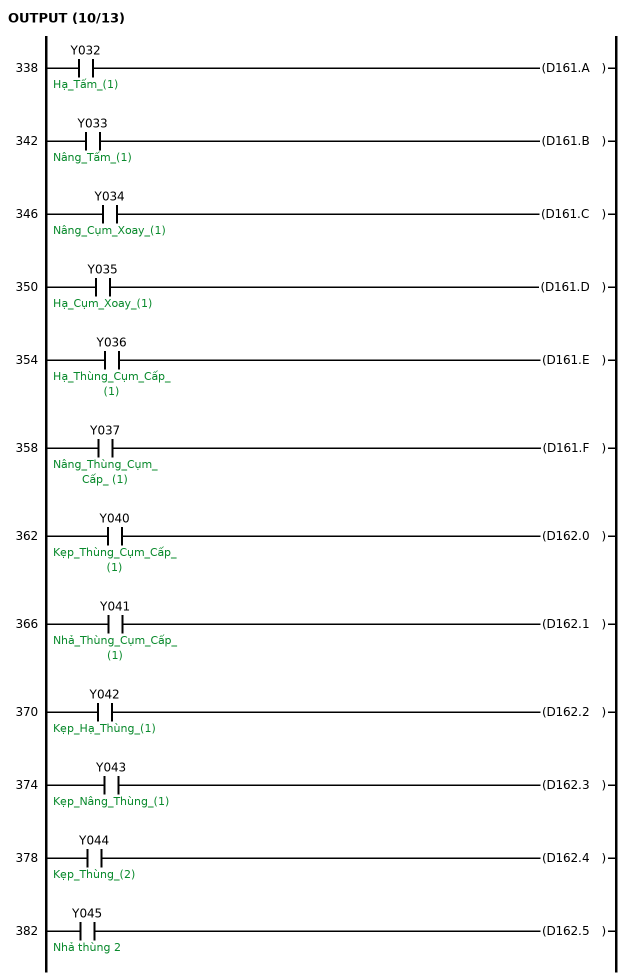
[picture p48: ladder of OUTPUT, rungs at steps 338 to 382]
338   LD      Y032  ; Hạ_Tấm_(1)
      OUT     D161.A
342   LD      Y033  ; Nâng_Tấm_(1)
      OUT     D161.B
346   LD      Y034  ; Nâng_Cụm_Xoay_(1)
      OUT     D161.C
350   LD      Y035  ; Hạ_Cụm_Xoay_(1)
      OUT     D161.D
354   LD      Y036  ; Hạ_Thùng_Cụm_Cấp_ (1)
      OUT     D161.E
358   LD      Y037  ; Nâng_Thùng_Cụm_Cấp_ (1)
      OUT     D161.F
362   LD      Y040  ; Kẹp_Thùng_Cụm_Cấp_(1)
      OUT     D162.0
366   LD      Y041  ; Nhả_Thùng_Cụm_Cấp_(1)
      OUT     D162.1
370   LD      Y042  ; Kẹp_Hạ_Thùng_(1)
      OUT     D162.2
374   LD      Y043  ; Kẹp_Nâng_Thùng_(1)
      OUT     D162.3
378   LD      Y044  ; Kẹp_Thùng_(2)
      OUT     D162.4
382   LD      Y045  ; Nhả thùng 2
      OUT     D162.5
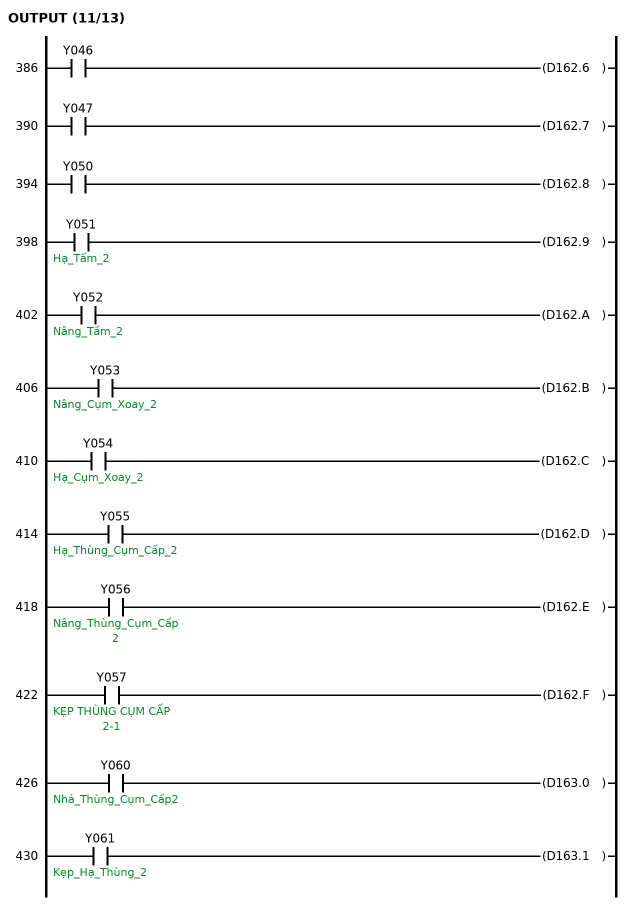
386   LD      Y046
      OUT     D162.6
390   LD      Y047
      OUT     D162.7
394   LD      Y050
      OUT     D162.8
398   LD      Y051  ; Hạ_Tấm_2
      OUT     D162.9
402   LD      Y052  ; Nâng_Tấm_2
      OUT     D162.A
406   LD      Y053  ; Nâng_Cụm_Xoay_2
      OUT     D162.B
410   LD      Y054  ; Hạ_Cụm_Xoay_2
      OUT     D162.C
414   LD      Y055  ; Hạ_Thùng_Cụm_Cấp_2
      OUT     D162.D
418   LD      Y056  ; Nâng_Thùng_Cụm_Cấp 2
      OUT     D162.E
422   LD      Y057  ; KẸP THÙNG CỤM CẤP 2-1
      OUT     D162.F
426   LD      Y060  ; Nhả_Thùng_Cụm_Cấp2
      OUT     D163.0
430   LD      Y061  ; Kẹp_Hạ_Thùng_2
      OUT     D163.1
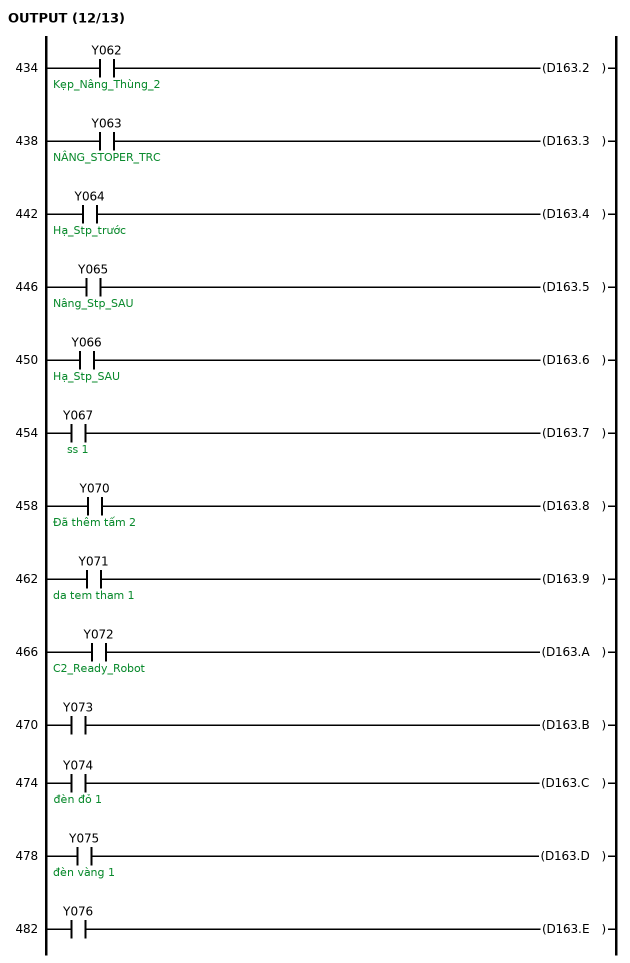
434   LD      Y062  ; Kẹp_Nâng_Thùng_2
      OUT     D163.2
438   LD      Y063  ; NÂNG_STOPER_TRC
      OUT     D163.3
442   LD      Y064  ; Hạ_Stp_trước
      OUT     D163.4
446   LD      Y065  ; Nâng_Stp_SAU
      OUT     D163.5
450   LD      Y066  ; Hạ_Stp_SAU
      OUT     D163.6
454   LD      Y067  ; ss 1
      OUT     D163.7
458   LD      Y070  ; Đã thêm tấm 2
      OUT     D163.8
462   LD      Y071  ; da tem tham 1
      OUT     D163.9
466   LD      Y072  ; C2_Ready_Robot
      OUT     D163.A
470   LD      Y073
      OUT     D163.B
474   LD      Y074  ; đèn đỏ 1
      OUT     D163.C
478   LD      Y075  ; đèn vàng 1
      OUT     D163.D
482   LD      Y076
      OUT     D163.E
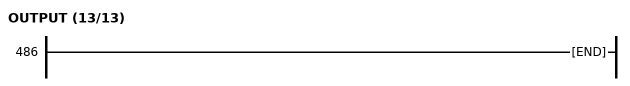
486   END
END_PROGRAM

PROGRAM PC_Ctrl
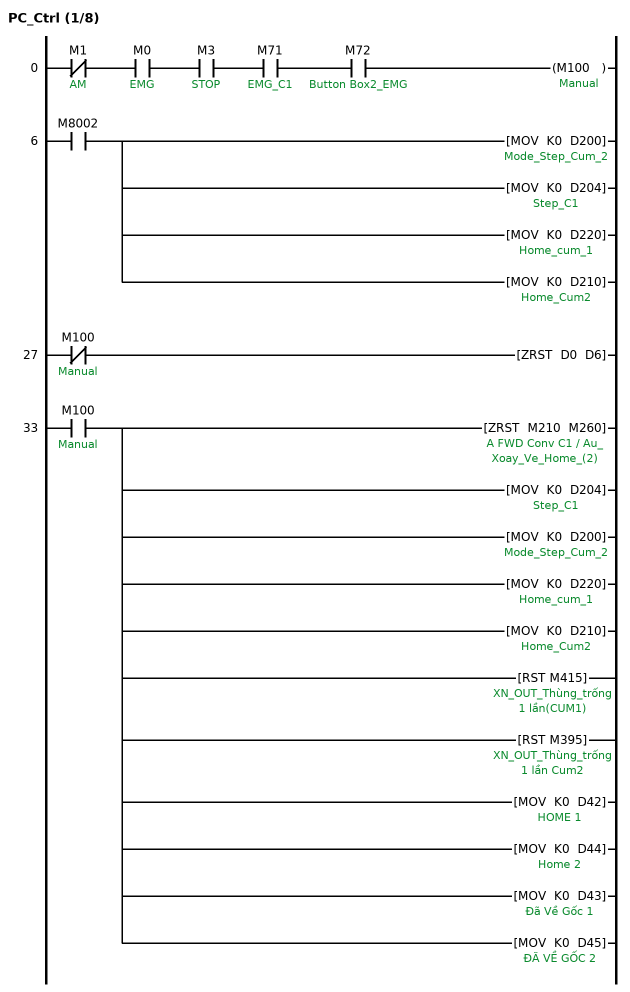
0     LDI     M1  ; AM
      AND     M0  ; EMG
      AND     M3  ; STOP
      AND     M71  ; EMG_C1
      AND     M72  ; Button Box2_EMG
      OUT     M100  ; Manual
6     LD      M8002
      MOV     K0 D200  ; Mode_Step_Cum_2
      MOV     K0 D204  ; Step_C1
      MOV     K0 D220  ; Home_cum_1
      MOV     K0 D210  ; Home_Cum2
27    LDI     M100  ; Manual
      ZRST    D0 D6
33    LD      M100  ; Manual
      ZRST    M210 M260  ; A FWD Conv C1 / Au_ Xoay_Ve_Home_(2)
      MOV     K0 D204
      MOV     K0 D200
      MOV     K0 D220
      MOV     K0 D210
      RST     M415  ; XN_OUT_Thùng_trống 1 lần(CUM1)
      RST     M395  ; XN_OUT_Thùng_trống 1 lần Cum2
      MOV     K0 D42  ; HOME 1
      MOV     K0 D44  ; Home 2
      MOV     K0 D43  ; Đã Về Gốc 1
      MOV     K0 D45  ; ĐÃ VỀ GỐC 2
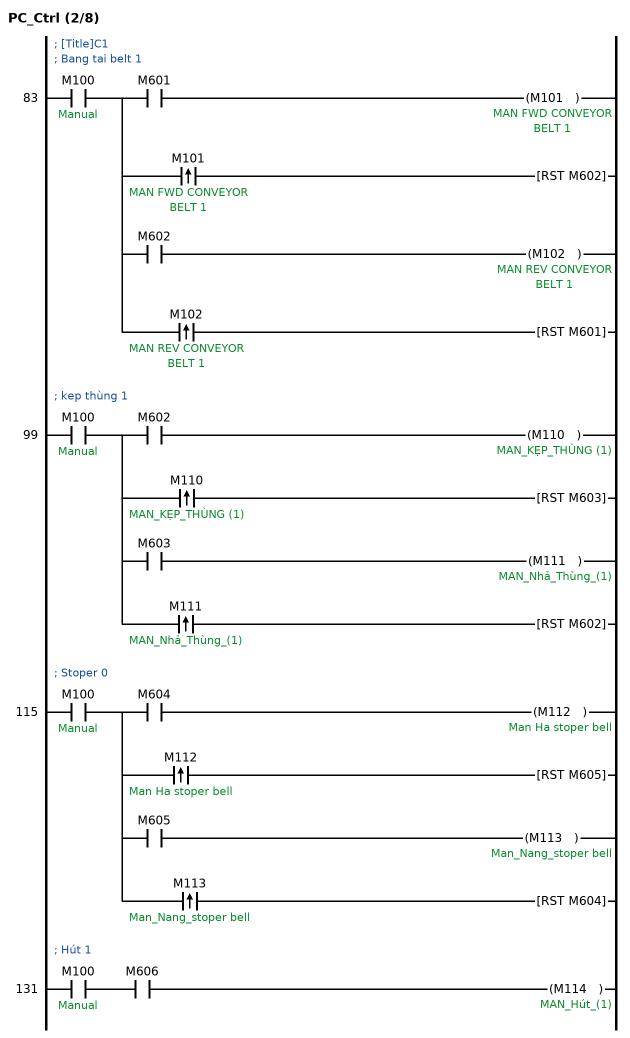
; [Title]C1
; Bang tai belt 1
83    LD      M100  ; Manual
      MPS
      AND     M601
      OUT     M101  ; MAN FWD CONVEYOR BELT 1
      MRD
      ANDP    M101  ; MAN FWD CONVEYOR BELT 1
      RST     M602
      MRD
      AND     M602
      OUT     M102  ; MAN REV CONVEYOR BELT 1
      MPP
      ANDP    M102  ; MAN REV CONVEYOR BELT 1
      RST     M601
; kep thùng 1
99    LD      M100  ; Manual
      MPS
      AND     M602
      OUT     M110  ; MAN_KẸP_THÙNG (1)
      MRD
      ANDP    M110  ; MAN_KẸP_THÙNG (1)
      RST     M603
      MRD
      AND     M603
      OUT     M111  ; MAN_Nhả_Thùng_(1)
      MPP
      ANDP    M111  ; MAN_Nhả_Thùng_(1)
      RST     M602
; Stoper 0
115   LD      M100  ; Manual
      MPS
      AND     M604
      OUT     M112  ; Man Ha stoper bell
      MRD
      ANDP    M112  ; Man Ha stoper bell
      RST     M605
      MRD
      AND     M605
      OUT     M113  ; Man_Nang_stoper bell
      MPP
      ANDP    M113  ; Man_Nang_stoper bell
      RST     M604
; Hút 1
131   LD      M100  ; Manual
      AND     M606
      OUT     M114  ; MAN_Hút_(1)
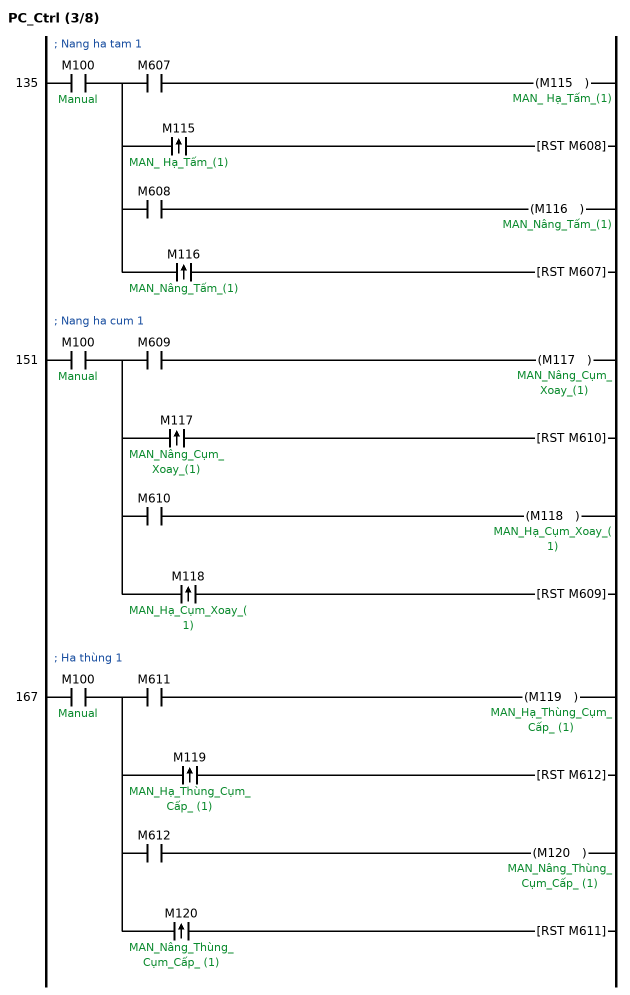
; Nang ha tam 1
135   LD      M100  ; Manual
      MPS
      AND     M607
      OUT     M115  ; MAN_ Hạ_Tấm_(1)
      MRD
      ANDP    M115  ; MAN_ Hạ_Tấm_(1)
      RST     M608
      MRD
      AND     M608
      OUT     M116  ; MAN_Nâng_Tấm_(1)
      MPP
      ANDP    M116  ; MAN_Nâng_Tấm_(1)
      RST     M607
; Nang ha cum 1
151   LD      M100  ; Manual
      MPS
      AND     M609
      OUT     M117  ; MAN_Nâng_Cụm_Xoay_(1)
      MRD
      ANDP    M117  ; MAN_Nâng_Cụm_Xoay_(1)
      RST     M610
      MRD
      AND     M610
      OUT     M118  ; MAN_Hạ_Cụm_Xoay_(1)
      MPP
      ANDP    M118  ; MAN_Hạ_Cụm_Xoay_(1)
      RST     M609
; Ha thùng 1
167   LD      M100  ; Manual
      MPS
      AND     M611
      OUT     M119  ; MAN_Hạ_Thùng_Cụm_Cấp_ (1)
      MRD
      ANDP    M119  ; MAN_Hạ_Thùng_Cụm_Cấp_ (1)
      RST     M612
      MRD
      AND     M612
      OUT     M120  ; MAN_Nâng_Thùng_Cụm_Cấp_ (1)
      MPP
      ANDP    M120  ; MAN_Nâng_Thùng_Cụm_Cấp_ (1)
      RST     M611
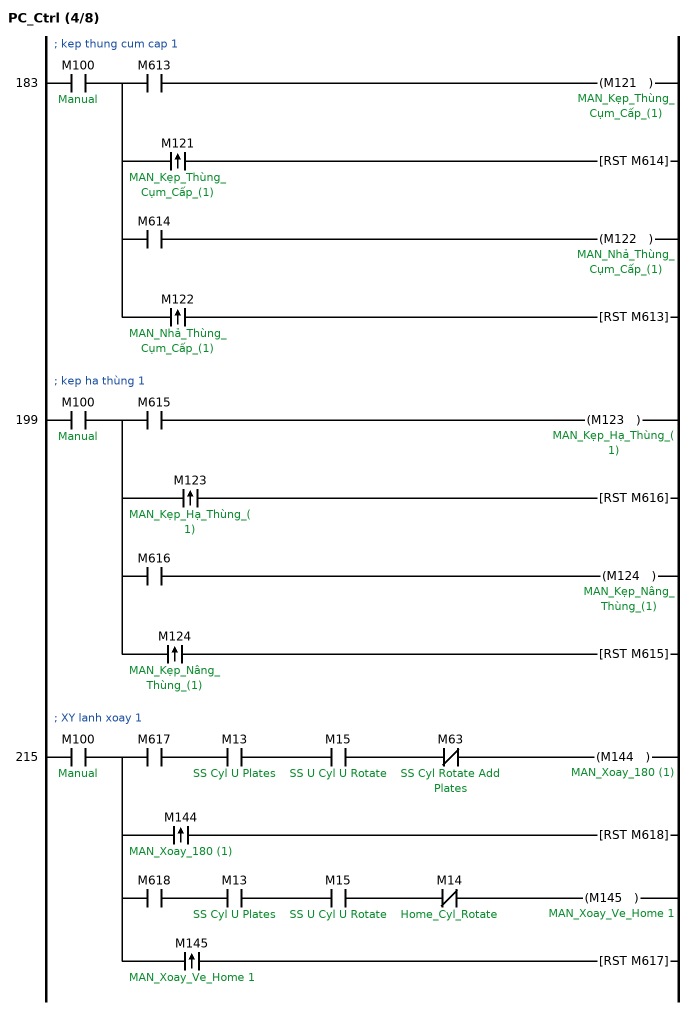
; kep thung cum cap 1
183   LD      M100  ; Manual
      MPS
      AND     M613
      OUT     M121  ; MAN_Kẹp_Thùng_Cụm_Cấp_(1)
      MRD
      ANDP    M121  ; MAN_Kẹp_Thùng_Cụm_Cấp_(1)
      RST     M614
      MRD
      AND     M614
      OUT     M122  ; MAN_Nhả_Thùng_Cụm_Cấp_(1)
      MPP
      ANDP    M122  ; MAN_Nhả_Thùng_Cụm_Cấp_(1)
      RST     M613
; kep ha thùng 1
199   LD      M100  ; Manual
      MPS
      AND     M615
      OUT     M123  ; MAN_Kẹp_Hạ_Thùng_(1)
      MRD
      ANDP    M123  ; MAN_Kẹp_Hạ_Thùng_(1)
      RST     M616
      MRD
      AND     M616
      OUT     M124  ; MAN_Kẹp_Nâng_Thùng_(1)
      MPP
      ANDP    M124  ; MAN_Kẹp_Nâng_Thùng_(1)
      RST     M615
; XY lanh xoay 1
215   LD      M100  ; Manual
      MPS
      AND     M617
      AND     M13  ; SS Cyl U Plates
      AND     M15  ; SS U Cyl U Rotate
      ANI     M63  ; SS Cyl Rotate Add Plates
      OUT     M144  ; MAN_Xoay_180 (1)
      MRD
      ANDP    M144  ; MAN_Xoay_180 (1)
      RST     M618
      MRD
      AND     M618
      AND     M13  ; SS Cyl U Plates
      AND     M15  ; SS U Cyl U Rotate
      ANI     M14  ; Home_Cyl_Rotate
      OUT     M145  ; MAN_Xoay_Ve_Home 1
      MPP
      ANDP    M145  ; MAN_Xoay_Ve_Home 1
      RST     M617
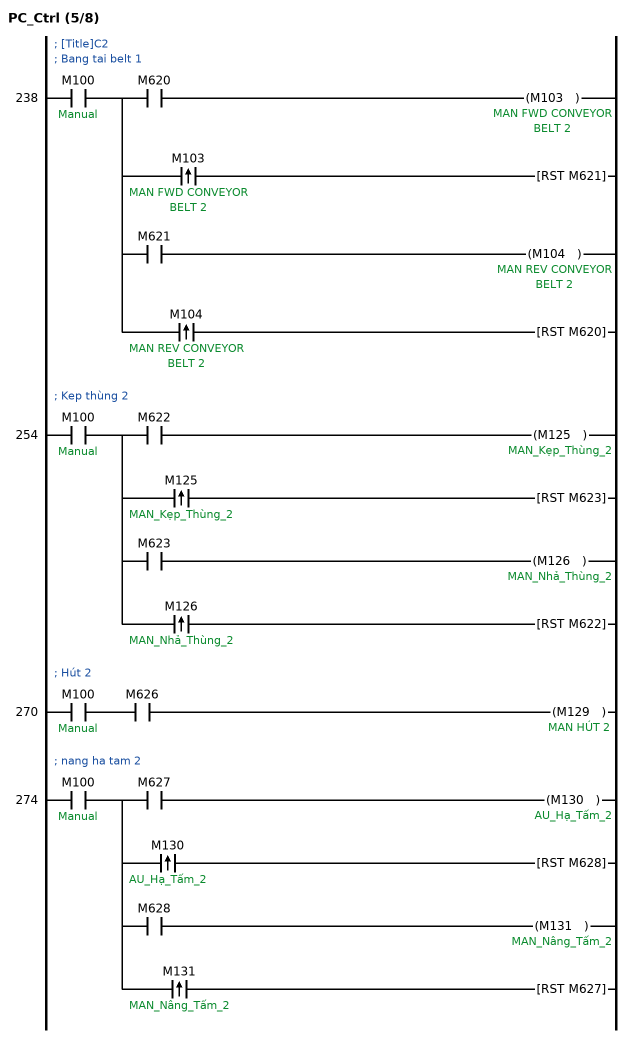
; [Title]C2
; Bang tai belt 1
238   LD      M100  ; Manual
      MPS
      AND     M620
      OUT     M103  ; MAN FWD CONVEYOR BELT 2
      MRD
      ANDP    M103  ; MAN FWD CONVEYOR BELT 2
      RST     M621
      MRD
      AND     M621
      OUT     M104  ; MAN REV CONVEYOR BELT 2
      MPP
      ANDP    M104  ; MAN REV CONVEYOR BELT 2
      RST     M620
; Kep thùng 2
254   LD      M100  ; Manual
      MPS
      AND     M622
      OUT     M125  ; MAN_Kẹp_Thùng_2
      MRD
      ANDP    M125  ; MAN_Kẹp_Thùng_2
      RST     M623
      MRD
      AND     M623
      OUT     M126  ; MAN_Nhả_Thùng_2
      MPP
      ANDP    M126  ; MAN_Nhả_Thùng_2
      RST     M622
; Hút 2
270   LD      M100  ; Manual
      AND     M626
      OUT     M129  ; MAN HÚT 2
; nang ha tam 2
274   LD      M100  ; Manual
      MPS
      AND     M627
      OUT     M130  ; AU_Hạ_Tấm_2
      MRD
      ANDP    M130  ; AU_Hạ_Tấm_2
      RST     M628
      MRD
      AND     M628
      OUT     M131  ; MAN_Nâng_Tấm_2
      MPP
      ANDP    M131  ; MAN_Nâng_Tấm_2
      RST     M627
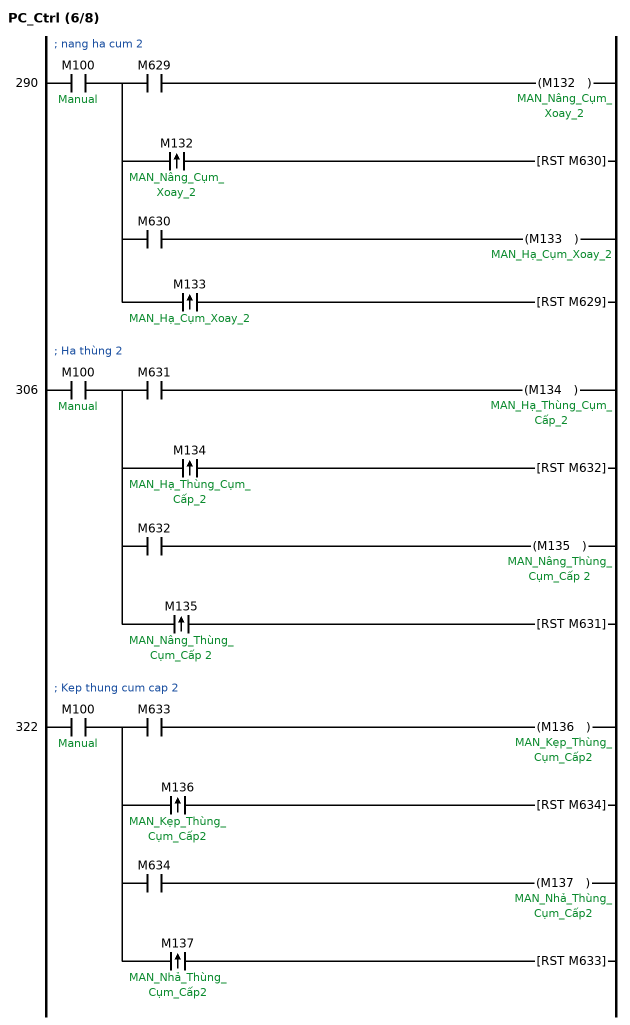
; nang ha cum 2
290   LD      M100  ; Manual
      MPS
      AND     M629
      OUT     M132  ; MAN_Nâng_Cụm_Xoay_2
      MRD
      ANDP    M132  ; MAN_Nâng_Cụm_Xoay_2
      RST     M630
      MRD
      AND     M630
      OUT     M133  ; MAN_Hạ_Cụm_Xoay_2
      MPP
      ANDP    M133  ; MAN_Hạ_Cụm_Xoay_2
      RST     M629
; Ha thùng 2
306   LD      M100  ; Manual
      MPS
      AND     M631
      OUT     M134  ; MAN_Hạ_Thùng_Cụm_Cấp_2
      MRD
      ANDP    M134  ; MAN_Hạ_Thùng_Cụm_Cấp_2
      RST     M632
      MRD
      AND     M632
      OUT     M135  ; MAN_Nâng_Thùng_Cụm_Cấp 2
      MPP
      ANDP    M135  ; MAN_Nâng_Thùng_Cụm_Cấp 2
      RST     M631
; Kep thung cum cap 2
322   LD      M100  ; Manual
      MPS
      AND     M633
      OUT     M136  ; MAN_Kẹp_Thùng_Cụm_Cấp2
      MRD
      ANDP    M136  ; MAN_Kẹp_Thùng_Cụm_Cấp2
      RST     M634
      MRD
      AND     M634
      OUT     M137  ; MAN_Nhả_Thùng_Cụm_Cấp2
      MPP
      ANDP    M137  ; MAN_Nhả_Thùng_Cụm_Cấp2
      RST     M633
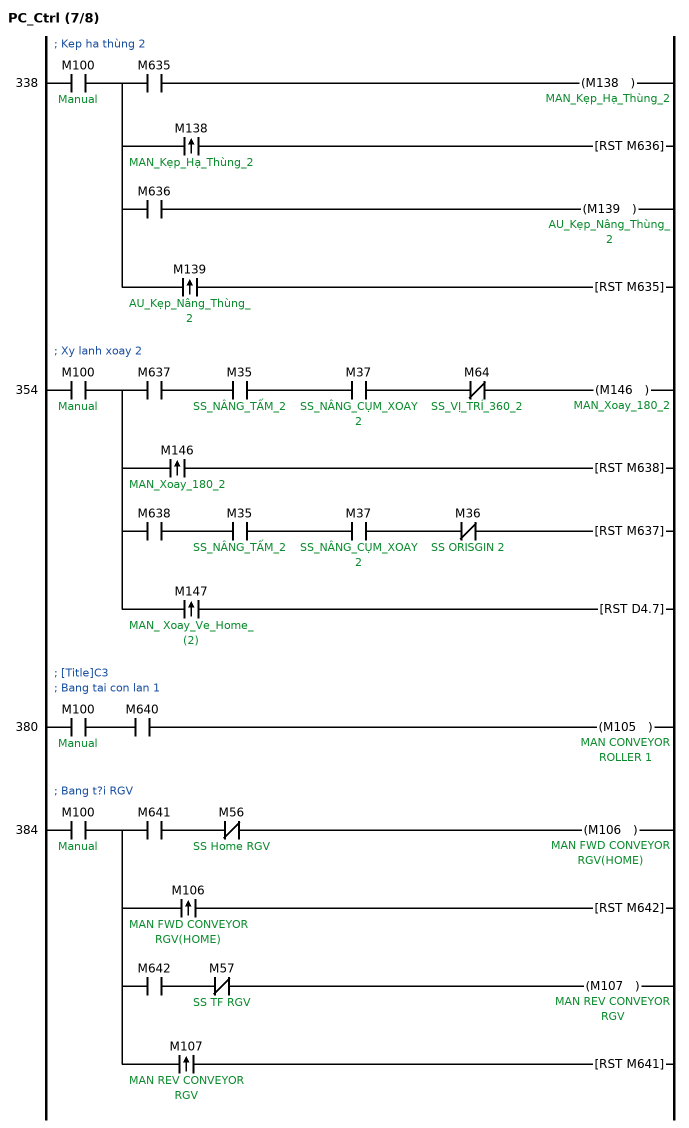
; Kep ha thùng 2
338   LD      M100  ; Manual
      MPS
      AND     M635
      OUT     M138  ; MAN_Kẹp_Hạ_Thùng_2
      MRD
      ANDP    M138  ; MAN_Kẹp_Hạ_Thùng_2
      RST     M636
      MRD
      AND     M636
      OUT     M139  ; AU_Kẹp_Nâng_Thùng_2
      MPP
      ANDP    M139  ; AU_Kẹp_Nâng_Thùng_2
      RST     M635
; Xy lanh xoay 2
354   LD      M100  ; Manual
      MPS
      AND     M637
      AND     M35  ; SS_NÂNG_TẤM_2
      AND     M37  ; SS_NÂNG_CỤM_XOAY 2
      ANI     M64  ; SS_VỊ_TRÍ_360_2
      OUT     M146  ; MAN_Xoay_180_2
      MRD
      ANDP    M146  ; MAN_Xoay_180_2
      RST     M638
      MRD
      AND     M638
      AND     M35  ; SS_NÂNG_TẤM_2
      AND     M37  ; SS_NÂNG_CỤM_XOAY 2
      ANI     M36  ; SS ORISGIN 2
      RST     M637
      MPP
      ANDP    M147  ; MAN_ Xoay_Ve_Home_(2)
      RST     D4.7
; [Title]C3
; Bang tai con lan 1
; 
380   LD      M100  ; Manual
      AND     M640
      OUT     M105  ; MAN CONVEYOR ROLLER 1
; Bang t?i RGV
384   LD      M100  ; Manual
      MPS
      AND     M641
      ANI     M56  ; SS Home RGV
      OUT     M106  ; MAN FWD CONVEYOR RGV(HOME)
      MRD
      ANDP    M106  ; MAN FWD CONVEYOR RGV(HOME)
      RST     M642
      MRD
      AND     M642
      ANI     M57  ; SS TF RGV
      OUT     M107  ; MAN REV CONVEYOR RGV
      MPP
      ANDP    M107  ; MAN REV CONVEYOR RGV
      RST     M641
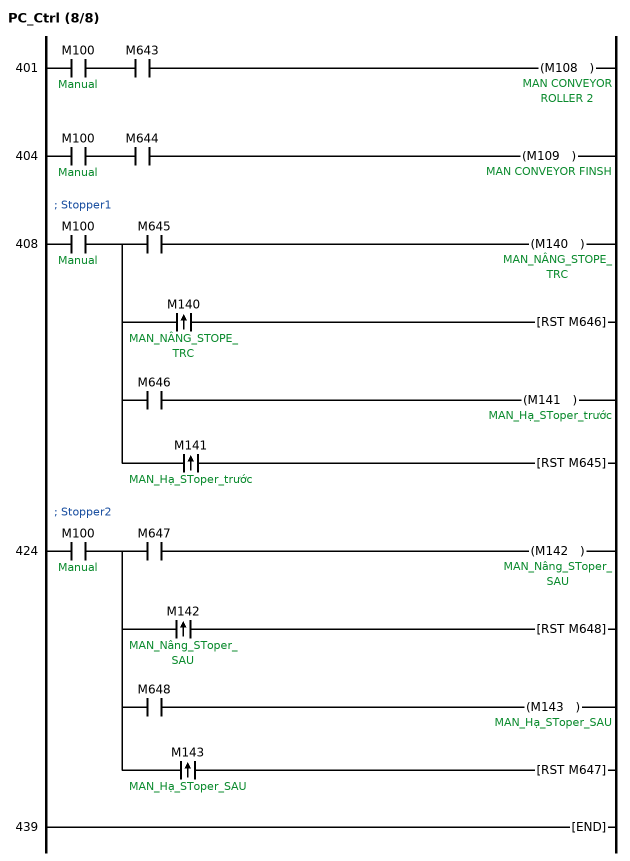
401   LD      M100  ; Manual
      AND     M643
      OUT     M108  ; MAN CONVEYOR ROLLER 2
404   LD      M100  ; Manual
      AND     M644
      OUT     M109  ; MAN CONVEYOR FINSH
; Stopper1
408   LD      M100  ; Manual
      MPS
      AND     M645
      OUT     M140  ; MAN_NÂNG_STOPE_TRC
      MRD
      ANDP    M140  ; MAN_NÂNG_STOPE_TRC
      RST     M646
      MRD
      AND     M646
      OUT     M141  ; MAN_Hạ_SToper_trước
      MPP
      ANDP    M141  ; MAN_Hạ_SToper_trước
      RST     M645
; Stopper2
424   LD      M100  ; Manual
      MPS
      AND     M647
      OUT     M142  ; MAN_Nâng_SToper_SAU
      MRD
      ANDP    M142  ; MAN_Nâng_SToper_SAU
      RST     M648
      MRD
      AND     M648
      OUT     M143  ; MAN_Hạ_SToper_SAU
      MPP
      ANDP    M143  ; MAN_Hạ_SToper_SAU
      RST     M647
439   END
END_PROGRAM

// device comments not shown above
M150  ; MAN 1
M151  ; MAN2
M180  ; HOME
M181  ; HOME 1
M182  ; HOME 2
M195  ; TG STOP
M196  ; NGAT HUT 1
M197  ; NGAT HUT 2
M198  ; TG TRA HANG 2
M199  ; TG TRA HANG 1
M200  ; AUTO
M203  ; Tạm dừng 1
M205  ; HMI_AUTO1
M206  ; HMI_AUTO2
M301  ; TG CHECK VỊ TRÍ LẤY TẤM 1
M302  ; TG CHECK GỐC 1
M303  ; Thêm tấm 1
M305  ; OFF HÚT 1
M306  ; TG TIMER DELAY STOPPER
M310  ; ATUO_SERVO 2 QUAY 180
M311  ; TG CHECK VỊ TRÍ LẤY TẤM 2
M312  ; TG CHECK GỐC 2
M313  ; Thêm tấm 2
M315  ; OFF HÚT 2
M322  ; SS hàng 1 tam (2) va da thêm tam
M326  ; Sansang hang 1 cum
M335  ; KHÓA TAY XOAY 2
M350  ; Req_Add_Plate_C1
M385  ; Home_cum2
M386  ; Bit_Home1
M397  ; Bit_XN_da_xoay_Manual(Cum2)
M399  ; Hang 2 tam
M410  ; Bit_XN_da_xoay_Manual(Cum2)
D1  ; Man_Device_Cum1
D2  ; MAN Device cum1
D3  ; Man Device cum2
D4  ; Man Device cum2
D5  ; MAN Device Cum2
D7  ; MAN HẠ THÙNG 1
D8  ; MAN KẸP THÙNG CỤM CẤP 1
D9  ; MAN KẸP HẠ THÙNG 1
D10  ; XY LANK XOAY1
D11  ; MAN CONVEYOR BELT 2
D12  ; MAN KẸP THÙNG 2
D13  ; MAN KẸP TẤM 2
D14  ; MAN HÚT 2
D15  ; MAN NÂNG HẠ TẤM 2-1
D16  ; MAN NÂNG HẠ CỤM 2
D17  ; MAN HẠ THÙNG 2
D18  ; MAN KẸP THÙNG CỤM CẤP 2
D19  ; MAN KẸP HẠ THÙNG 2
D20  ; XY LANK XOAY2
D21  ; MAN CONVEYOR ROLLER 1
D22  ; MAN CONVEYOR RGV
D23  ; MAN CONVEYOR ROLLER 2
D24  ; MAN CONVEYOR FINSH
D25  ; MAN STOPPER 1
D26  ; MAN STOPPER 2
D27  ; PC START
D28  ; PC STOP
D29  ; PC Reset
D40  ; Đổi Model 2 tầng cụm 2
D47  ; TẠM DỪNG 2
D49  ; KHÓA TAY XOAY 2
D51  ; HMI_LIGHT AUTO1
D52  ; HMI_LIGHT AUTO2
D53  ; AU/MAN 1
D54  ; AU/MAN2
D55  ; HMI_NÚT ĐẦY THÙNG 1
D56  ; HMI_ĐẦY THÙNG 2
D57  ; XÁC NHẬN ĐÃ THÊM TẤM 1
D58  ; XÁC NHẬN ĐÃ CẤP THÙNG 1
D59  ; XÁC NHẬN ĐÃ THÊM TẤM 2
D60  ; XÁC NHẬN ĐÃ THAY THÙNG 2
D101  ; LỖI AN TOÀN CỤM 1
D102  ; LỖI AN TOÀN CỤM 2
D230  ; Out Product C1
D252  ; Hang 1 or 2 ( cum1)
T52  ; Timer_ko_Co_hang_2
T160  ; timer_Ngatthemtam
T161  ; test robot báo đầy thùng(2)
T162  ; test robot báo thêm tấm 1
T166  ; Timer ss dung bang tai 2
T168  ; Timer home 2 bang tai
